// TwinCAT 3 PLC project FanucIntegrationV2
// ProgramVersion: 3.1.4026.26
// libraries:
//   Tc2_Standard, * (Beckhoff Automation GmbH)
//   Tc2_System, * (Beckhoff Automation GmbH)
//   FanucSimpleLib,2.1.0.0,Beckhoff Automation IL
// project tree:
//   DUTs/ E_FanucCstopiState.TcDUT, E_FanucEnableState.TcDUT, E_FanucFaultResetState.TcDUT, E_FanucHomingState.TcDUT, E_FanucStartProgramState.TcDUT, ST_FanucControl.TcDUT, ST_FanucStatus.TcDUT
//   GVLs/ GVL_Fanuc.TcGVL (not stored)
//   / PlcTask.TcTTO
//   POUs/ FB_FanucControl.TcPOU, FB_FanucCycleStop.TcPOU, FB_FanucEnable.TcPOU, FB_FanucFaultReset.TcPOU, FB_FanucHoming.TcPOU, FB_FanucSpeedOverride.TcPOU, FB_FanucStartProgram.TcPOU, FB_FanucStatus.TcPOU, MAIN.TcPOU
// real-time tasks:
//   TASK PlcTask: cycle T#10ms, priority 20, ADS port 350

CONFIGURATION FanucIntegrationV2
    RESOURCE PLC ON TwinCAT3
        TASK PlcTask(INTERVAL := T#10ms, PRIORITY := 20);
        PROGRAM MAIN WITH PlcTask : MAIN;
    END_RESOURCE
END_CONFIGURATION

// ---- DUTs/E_FanucCstopiState.TcDUT
// States used by FB_FanucCycleStop.

TYPE E_FanucCstopiState :
(
	Idle	:= 0, // Waits for a rising edge of bStart.
	Pulsing	:= 1, // Generates the CSTOPI pulse for tCycleStopPulse.
	Done	:= 2 // Sets bDone for one PLC scan to confirm pulse completion, then returns to Idle.
);
END_TYPE

// ---- DUTs/E_FanucEnableState.TcDUT
// States used by FB_FanucEnable.

TYPE E_FanucEnableState :
(
	Idle			:= 0, // ENBL is FALSE; waits for all enable permissives and bExtStart = FALSE.
	ClearFault		:= 1, // Waits for bFault = FALSE; this state does not generate FAULT_RESET.
	CheckTP			:= 3, // Waits for bTP_Enabled = FALSE before proceeding to WaitReady.
	WaitReady		:= 4, // Waits for bCmd_Enabled AND bSystem_Ready within tReadyTimeout.
	Ready			:= 5, // Sets bReady and accepts START edges while monitoring faults and interlocks.
	Paused			:= 6, // Waits for bExtHold = TRUE and bMotion_Held = FALSE before returning to Ready.
	EmergencyStop	:= 7, // Waits for bExtIMSTP = TRUE before returning through ClearFault.
	SafeSpeed		:= 8, // Waits for bExtSFSPD = TRUE before returning to Ready or Paused.
	Error			:= 99 // Sets bError and removes ENBL; bEnable = FALSE returns to Idle.
);
END_TYPE

// ---- DUTs/E_FanucFaultResetState.TcDUT
// States used by FB_FanucFaultReset.

TYPE E_FanucFaultResetState :
(
	Idle		:= 0, // Waits for a rising edge of bReset.
	SendPulse	:= 1, // Generates the FAULT_RESET pulse for tResetPulse.
	WaitClear	:= 2, // Waits for bFault = FALSE within tFaultTimeout after the pulse.
	Done		:= 3, // Sets bDone for one PLC scan, then returns to Idle.
	Error		:= 99 // Sets bError; bReset = FALSE returns to Idle.
);
END_TYPE

// ---- DUTs/E_FanucHomingState.TcDUT
// States used by FB_FanucHoming.

TYPE E_FanucHomingState :
(
	Idle			:= 0, // Waits for a rising edge of bStart while bReady = TRUE.
	RequestHome		:= 1, // Generates the HOME pulse for tHomePulse while bReady remains TRUE.
	WaitComplete	:= 2, // Waits for bAt_Home = TRUE within tHomingTimeout while bReady remains TRUE.
	Done			:= 3, // Sets bDone for one PLC scan, then returns to Idle.
	Error			:= 99 // Sets bError; bStart = FALSE returns to Idle.
);
END_TYPE

// ---- DUTs/E_FanucStartProgramState.TcDUT
// States used by FB_FanucStartProgram.

TYPE E_FanucStartProgramState :
(
	Idle	:= 0, // Waits for a rising edge of bStart while bReady = TRUE, then validates nProgram.
	Pulsing	:= 1, // Generates the selected RSR pulse for tProgramPulse and monitors its ACK.
	WaitAck	:= 2, // Waits for a fresh matching ACK within tAckTimeout after the pulse.
	Done	:= 3, // Sets bDone for one PLC scan to confirm acknowledgement, then returns to Idle.
	Error	:= 99 // Sets bError; bStart = FALSE returns to Idle.
);
END_TYPE

// ---- DUTs/ST_FanucControl.TcDUT
// FANUC command signals encoded by FB_FanucControl.
// UI numbers refer to robot inputs; aDO references refer to PLC output bytes.

TYPE ST_FanucControl :
STRUCT
	// Control byte 0: UI[1..8].
	IMSTP 		: BOOL; // aDO[0].0 | UI[1] *IMSTP: TRUE releases the request; FALSE requests an immediate stop.
	Hold		: BOOL; // aDO[0].1 | UI[2] *HOLD: TRUE releases the request; FALSE requests a hold.
	SFSPD		: BOOL; // aDO[0].2 | UI[3] *SFSPD: TRUE releases the request; FALSE asserts the SFSPD request.
	Cycle_stop	: BOOL; // aDO[0].3 | UI[4] CSTOPI: Cycle Stop command; effect depends on FANUC configuration.
	Fault_Reset	: BOOL; // aDO[0].4 | UI[5] FAULT_RESET: command pulse to reset clearable robot faults.
	Start		: BOOL; // aDO[0].5 | UI[6] START: start/resume command signal.
	Home		: BOOL; // aDO[0].6 | UI[7] HOME: command signal for the configured homing macro.
	Enable		: BOOL; // aDO[0].7 | UI[8] ENBL: TRUE enables motion subject to the remaining robot conditions.

	// Control byte 1: RSR selections or PNS bits, depending on robot mode.
	Start_Program1	: BOOL; // aDO[1].0 | UI[9]: RSR1 request or PNS bit 0.
	Start_Program2	: BOOL; // aDO[1].1 | UI[10]: RSR2 request or PNS bit 1.
	Start_Program3	: BOOL; // aDO[1].2 | UI[11]: RSR3 request or PNS bit 2.
	Start_Program4	: BOOL; // aDO[1].3 | UI[12]: RSR4 request or PNS bit 3.
	Start_Program5	: BOOL; // aDO[1].4 | UI[13]: RSR5 request or PNS bit 4.
	Start_Program6	: BOOL; // aDO[1].5 | UI[14]: RSR6 request or PNS bit 5.
	Start_Program7	: BOOL; // aDO[1].6 | UI[15]: RSR7 request or PNS bit 6.
	Start_Program8	: BOOL; // aDO[1].7 | UI[16]: RSR8 request or PNS bit 7.

	// Control byte 2: PNS command signals.
	PNS_Strobe	: BOOL; // aDO[2].0 | UI[17] PNSTROBE: strobe for PNS program selection.
	Prod_Start	: BOOL; // aDO[2].1 | UI[18] PROD_START: execution request for the selected PNS program.

	// Control byte 3: application-configured speed override.
	Override : BYTE; // aDO[3] | Speed-override command in percent; map to the configured FANUC Group Input.
END_STRUCT
END_TYPE

// ---- DUTs/ST_FanucStatus.TcDUT
// FANUC feedback signals decoded by FB_FanucStatus.
// UO numbers refer to robot outputs; aDI references refer to PLC input bytes.

TYPE ST_FanucStatus :
STRUCT
	// Status byte 0: UO[1..8].
	bCmd_Enabled	: BOOL; // aDI[0].0 | UO[1] CMDENBL: TRUE when the robot reports command enable.
	bSystem_Ready	: BOOL; // aDI[0].1 | UO[2] SYSRDY: TRUE when the robot reports system ready.
	bPrg_Running	: BOOL; // aDI[0].2 | UO[3] PROGRUN: TRUE when the robot reports program execution.
	bPrg_Paused		: BOOL; // aDI[0].3 | UO[4] PAUSED: TRUE when the robot reports a paused program.
	bMotion_Held	: BOOL; // aDI[0].4 | UO[5] HELD: TRUE when the robot reports motion held.
	bFault			: BOOL; // aDI[0].5 | UO[6] FAULT: TRUE when the robot reports a fault.
	bAt_Home		: BOOL; // aDI[0].6 | UO[7] ATPERCH: TRUE at the configured reference position used as Home.
	bTP_Enabled		: BOOL; // aDI[0].7 | UO[8] TPENBL: TRUE when the teach pendant is enabled.

	// Status byte 1: UO[9..10].
	bBatteryAlarm	: BOOL; // aDI[1].0 | UO[9] BATALM: TRUE when the robot reports a battery alarm.
	bBusy			: BOOL; // aDI[1].1 | UO[10] BUSY: robot busy indication; separate from individual FB busy outputs.

	// Status byte 2: RSR acknowledgements or PNS selection feedback.
	bProg_Start1ACK	: BOOL; // aDI[2].0 | UO[11]: RSR1 acknowledgement or SNO1 in PNS mode.
	bProg_Start2ACK	: BOOL; // aDI[2].1 | UO[12]: RSR2 acknowledgement or SNO2 in PNS mode.
	bProg_Start3ACK	: BOOL; // aDI[2].2 | UO[13]: RSR3 acknowledgement or SNO3 in PNS mode.
	bProg_Start4ACK	: BOOL; // aDI[2].3 | UO[14]: RSR4 acknowledgement or SNO4 in PNS mode.
	bProg_Start5ACK	: BOOL; // aDI[2].4 | UO[15]: RSR5 acknowledgement or SNO5 in PNS mode.
	bProg_Start6ACK	: BOOL; // aDI[2].5 | UO[16]: RSR6 acknowledgement or SNO6 in PNS mode.
	bProg_Start7ACK	: BOOL; // aDI[2].6 | UO[17]: RSR7 acknowledgement or SNO7 in PNS mode.
	bProg_Start8ACK	: BOOL; // aDI[2].7 | UO[18]: RSR8 acknowledgement or SNO8 in PNS mode.
END_STRUCT
END_TYPE

// ---- POUs/MAIN.TcPOU
PROGRAM MAIN
VAR
	// ---------- Core robot interface (library FBs) ----------
	fbStatus			: FB_FanucStatus;			// DI0 byte array → stStatus struct
	fbControl			: FB_FanucControl;			// stControl struct → DO0 byte array
	fbEnable			: FB_FanucEnable;			// Enable sequence state machine
	fbFaultReset		: FB_FanucFaultReset;		// Fault reset pulse – FAULT_RESET (UI[5])
	fbStartProgram		: FB_FanucStartProgram;		// Program start – RSR (UI[9..16])
	fbCycleStop			: FB_FanucCycleStop;		// Cycle Stop – CSTOPI (UI[4])
	fbHoming			: FB_FanucHoming;			// Homing sequence – HOME (UI[7])
	stStatus			: ST_FanucStatus;			// Live robot status (inputs)
	stControl			: ST_FanucControl;			// Combined control command (outputs)
	fbSpeedOverride		: FB_FanucSpeedOverride;	// Writes byOverwrite value to GI[25..33] via stControl

	// ---------- Enable command ----------
	bEnableRobot		: BOOL;	// Set TRUE to start enable sequence

	// ---------- External interlock signals ----------
	bExtIMSTP			: BOOL;		// Normally closed: FALSE = software E-stop
	bExtHold			: BOOL;		// Normally closed: FALSE = pause/hold robot
	bExtSFSPD			: BOOL;		// Normally closed: FALSE = safe-speed limit active
	bExtStart			: BOOL;		// Rising edge triggers a 20 ms START pulse when Ready

	// ---------- Homing ----------
	bStartHome			: BOOL;		// Rising edge: start homing sequence (gated by bReady)

	// ---------- Program start ----------
	bStartProgram		: BOOL;		// Rising edge: start nProgram (gated by bReady)
	nProgram			: INT := 1;	// Program to start: 1..8 (RSR)

	// ---------- Cycle stop ----------
	bCycleStop			: BOOL;		// Rising edge: send CSTOPI cycle-stop command

	// ---------- Fault reset ----------
	bFaultReset			: BOOL;		// Rising edge: send FAULT_RESET pulse (UI[5])

	// ---------- Speed override ----------
	byOverwrite			: BYTE;		// Value sent to GI[25..33] via fbSpeedOverride (0–100)
	
END_VAR

// 1. Read status – always first
fbStatus(aDI := GVL_Fanuc.DI0, stStatus => stStatus);

// 2. Enable sequence (outputs stControl; other FBs stamp into it below)
fbEnable(
    bEnable		:= bEnableRobot,
    stStatus	:= stStatus,
    bExtIMSTP	:= bExtIMSTP,   // Wire from: NOT bSoftEStop
    bExtHold	:= bExtHold,    // Wire from: NOT bPauseButton
    bExtSFSPD	:= bExtSFSPD,   // Wire from: bFenceOK / area scanner
    bExtStart 	:= bExtStart,   // Wire from: HMI start button
	tReadyTimeout := T#5S,
	bReady=> , 
	bError=> , 
	bTPWarning=> , 
	eState=> , 
    stControl => stControl);
	
// 3. Homing
fbHoming(
    bStart    := bStartHome,
    bReady    := fbEnable.bReady,
	tHomingTimeout := T#15S, 
    stStatus  := stStatus,
    stControl := stControl,
	bBusy=> , 
	bDone=> , 
	bError=> , 
	eState=> );
	
// 4. Program start 
fbStartProgram(
	bStart		:= bStartProgram, 
	nProgram	:= nProgram , 
	bReady		:= fbEnable.bReady, 
	tAckTimeout	:= T#2S , 
	stStatus	:= stStatus, 
	stControl	:= stControl, 
	bRequestActive=> , 
	bDone=> , 
	bError=> , 
	eState=> );
	
// 5. Cycle stop
fbCycleStop(
	bStart:= bCycleStop, 
	tCycleStopPulse:= T#20MS, 
	stControl:= stControl, 
	bBusy=> , 
	bDone=> , 
	eState=> );
	
// 6. Fault reset (call when fbEnable.eState = ClearFault and operator requests)
fbFaultReset(
    bReset    := bFaultReset,
    stStatus  := stStatus,
    stControl := stControl);

// 7. Control robot speed via Overwrite
fbSpeedOverride(
	nOverwrite:= byOverwrite ,
	stControl:= stControl ,
	bError=>,
	nActual=>);
	
// 8. Write outputs – always last
fbControl(aDO := GVL_Fanuc.DO0, stControl := stControl);

END_PROGRAM

// ---- POUs/FB_FanucStatus.TcPOU
// Maps the FANUC input bytes to robot-status signals.
// Call every PLC scan before status-dependent logic.

FUNCTION_BLOCK FB_FanucStatus

VAR_IN_OUT
	aDI : ARRAY[0..15] OF BYTE; // Hardware-linked input bytes; pass GVL_Fanuc.DI0. Reads bytes 0..2.
END_VAR

VAR_OUTPUT
	stStatus : ST_FanucStatus; // Robot-status signals decoded from aDI during this call.
END_VAR


// Status Byte 0  (aDI[0])  -  UO[1..8]
stStatus.bCmd_Enabled  := aDI[0].0;   // UO[1]  CMDENBL  – command enable
stStatus.bSystem_Ready := aDI[0].1;   // UO[2]  SYSRDY   – servo powered, no alarm
stStatus.bPrg_Running  := aDI[0].2;   // UO[3]  PROGRUN  – program in execution
stStatus.bPrg_Paused   := aDI[0].3;   // UO[4]  PAUSED   – program on hold
stStatus.bMotion_Held  := aDI[0].4;   // UO[5]  HELD     – HOLD button/signal active
stStatus.bFault        := aDI[0].5;   // UO[6]  FAULT    – alarm preventing execution
stStatus.bAt_Home      := aDI[0].6;   // UO[7]  ATPERCH  – robot at reference position 1
stStatus.bTP_Enabled   := aDI[0].7;   // UO[8]  TPENBL   – teach pendant enable switch ON

// Status Byte 1  (aDI[1])  -  UO[9..10]
stStatus.bBatteryAlarm := aDI[1].0;   // UO[9]  BATALM   – controller battery low
stStatus.bBusy         := aDI[1].1;   // UO[10] BUSY     – program executing or TP busy

// Status Byte 2  (aDI[2])  -  UO[11..18]  RSR ACK / SNO
stStatus.bProg_Start1ACK := aDI[2].0; // UO[11] ACK1/SNO1
stStatus.bProg_Start2ACK := aDI[2].1; // UO[12] ACK2/SNO2
stStatus.bProg_Start3ACK := aDI[2].2; // UO[13] ACK3/SNO3
stStatus.bProg_Start4ACK := aDI[2].3; // UO[14] ACK4/SNO4
stStatus.bProg_Start5ACK := aDI[2].4; // UO[15] ACK5/SNO5
stStatus.bProg_Start6ACK := aDI[2].5; // UO[16] ACK6/SNO6
stStatus.bProg_Start7ACK := aDI[2].6; // UO[17] ACK7/SNO7
stStatus.bProg_Start8ACK := aDI[2].7; // UO[18] ACK8/SNO8

END_FUNCTION_BLOCK

// ---- POUs/FB_FanucControl.TcPOU
// Maps the FANUC control signals to the output bytes.
// Call every PLC scan after all FANUC command FBs.

FUNCTION_BLOCK FB_FanucControl

VAR_IN_OUT
	aDO : ARRAY[0..15] OF BYTE; // Hardware-linked output bytes; pass GVL_Fanuc.DO0. Writes bytes 0..3.
END_VAR

VAR_INPUT
	stControl : ST_FanucControl; // Combined FANUC commands to encode into aDO.
END_VAR


// Control Byte 0  (aDO[0])  -  UI[1..8]
aDO[0].0 := stControl.IMSTP;        // UI[1]  *IMSTP       NC – hold TRUE; FALSE = software E-stop
aDO[0].1 := stControl.Hold;         // UI[2]  *HOLD        NC – hold TRUE; FALSE = decelerate & pause
aDO[0].2 := stControl.SFSPD;        // UI[3]  *SFSPD       NC – hold TRUE; FALSE = safe-speed limit
aDO[0].3 := stControl.Cycle_stop;   // UI[4]  CSTOPI       pulse to stop/abort current cycle
aDO[0].4 := stControl.Fault_Reset;  // UI[5]  FAULT_RESET  pulse to reset clearable alarms
aDO[0].5 := stControl.Start;        // UI[6]  START        falling-edge resumes paused program
aDO[0].6 := stControl.Home;         // UI[7]  HOME         macro use only
aDO[0].7 := stControl.Enable;       // UI[8]  ENBL         NC – hold TRUE; FALSE = disable all motion

// Control Byte 1  (aDO[1])  -  UI[9..16]  RSR / PNS
aDO[1].0 := stControl.Start_Program1; // UI[9]  RSR1 / PNS bit 0
aDO[1].1 := stControl.Start_Program2; // UI[10] RSR2 / PNS bit 1
aDO[1].2 := stControl.Start_Program3; // UI[11] RSR3 / PNS bit 2
aDO[1].3 := stControl.Start_Program4; // UI[12] RSR4 / PNS bit 3
aDO[1].4 := stControl.Start_Program5; // UI[13] RSR5 / PNS bit 4
aDO[1].5 := stControl.Start_Program6; // UI[14] RSR6 / PNS bit 5
aDO[1].6 := stControl.Start_Program7; // UI[15] RSR7 / PNS bit 6
aDO[1].7 := stControl.Start_Program8; // UI[16] RSR8 / PNS bit 7

// Control Byte 2  (aDO[2])  -  UI[17..18]
aDO[2].0 := stControl.PNS_Strobe;                   // UI[17] reserved
aDO[2].1 := stControl.Prod_Start;   // UI[18] PROD_START – triggers PNS program execution

// Control Byte 3  (aDO[3])  -  GI[25..33] user-defined output
aDO[3] := stControl.Override;

END_FUNCTION_BLOCK

// ---- POUs/FB_FanucEnable.TcPOU
// Controls the FANUC remote-enable sequence and START pulse.
// External IMSTP, HOLD, and SFSPD signals pass through in every state.
// Fault reset is handled separately by FB_FanucFaultReset.

FUNCTION_BLOCK FB_FanucEnable

VAR_INPUT
	bEnable		: BOOL; // TRUE requests enabling; FALSE returns the FB to Idle and clears its error.
	stStatus	: ST_FanucStatus; // Live robot-status signals from FB_FanucStatus.

	bExtIMSTP	: BOOL; // IMSTP permissive: TRUE releases the request; FALSE requests an immediate stop.
	bExtHold	: BOOL; // HOLD permissive: TRUE releases the request; FALSE requests a hold.
	bExtSFSPD	: BOOL; // SFSPD permissive: TRUE releases the request; FALSE asserts the SFSPD request.

	bExtStart	: BOOL; // Rising edge requests a START pulse while Ready; must be FALSE to begin enabling.
	tReadyTimeout	: TIME := T#5S; // Maximum time in WaitReady for bCmd_Enabled AND bSystem_Ready.
END_VAR

VAR_OUTPUT
	bReady		: BOOL; // TRUE while the enable state machine is in Ready.
	bError		: BOOL; // TRUE in Error after a ready timeout or invalid state; cleared by bEnable = FALSE.
	bTPWarning	: BOOL; // TRUE while in CheckTP and the teach pendant is enabled.
	eState		: E_FanucEnableState; // Current state exposed for diagnostics and HMI.
	stControl	: ST_FanucControl; // Control structure; this FB writes Enable, IMSTP, Hold, SFSPD, and Start.
END_VAR

VAR
	eCurrentState : E_FanucEnableState := E_FanucEnableState.Idle; // Internal state used by the sequence.
	bEnablePermissivesOk : BOOL; // TRUE when bEnable, bExtIMSTP, bExtHold, and bExtSFSPD are all TRUE.
	tonReadyTimeout : TON; // Measures the time spent waiting in WaitReady.
	rtExtStart : R_TRIG; // Detects the FALSE-to-TRUE transition of bExtStart.
	bStartPulseActive : BOOL; // Latches the START pulse until its timer expires or Ready is lost.
	tonStartPulse : TON; // Measures the active START pulse duration.
END_VAR

VAR CONSTANT
	tStartPulse : TIME := T#20MS; // Requested duration of the START output pulse on UI[6].
END_VAR

(*
    FB_FanucEnable

    Purpose
    -------
    Controls the FANUC remote-enable state machine and produces
    the required UI control signals.

    Enable sequence
    ---------------

        Idle
          |
          | bEnable
          | + all interlocks OK
          | + bExtStart released
          v
        ClearFault
          |
          | bFault = FALSE
          v
        CheckTP
          |
          | TP disabled
          v
        WaitReady
          |
          | CMDENBL + SYSRDY
          v
        Ready


    Enable permissives
    ------------------
    The enable sequence requires:

        bEnable
        bExtIMSTP
        bExtHold
        bExtSFSPD

    These are combined internally as:

        bEnablePermissivesOk

    bExtStart is NOT an enable permissive.

    Start is a momentary command and is handled independently.


    ClearFault
    ----------
    This FB does NOT generate FAULT_RESET.

    While bFault remains TRUE, the state remains ClearFault.

    Use FB_FanucFaultReset externally to reset the FANUC fault.
    Once stStatus.bFault becomes FALSE, this FB automatically
    proceeds to CheckTP.


    Start behavior
    --------------
    bExtStart must be FALSE before the enable sequence can begin.

    Once Ready, an actual FALSE -> TRUE edge of bExtStart generates
    a tStartPulse pulse on stControl.Start.

    A Start edge occurring before Ready is ignored.

    If bExtStart is already TRUE when the robot enters Ready,
    no Start pulse is generated. It must first return FALSE and
    then receive a new rising edge.


    NC signal behavior
    ------------------
    Option A: passive while disabled.

    Idle / Error:
        ENBL  = FALSE
        IMSTP = TRUE
        HOLD  = TRUE
        SFSPD = TRUE

    Active states:
        ENBL  = TRUE
        IMSTP = bExtIMSTP
        HOLD  = bExtHold
        SFSPD = bExtSFSPD


    Error reset
    -----------
    To leave Error:

        bEnable := FALSE

    The FB then returns to Idle. A subsequent TRUE starts a new
    enable sequence.
*)

// Enable permissives
// ============================================================================
//
// These signals determine whether the robot is allowed to proceed through
// the enable sequence.
//
// bExtStart is intentionally NOT included.
// Start is a command, not a permissive.
//
bEnablePermissivesOk := bEnable AND bExtIMSTP AND bExtHold AND bExtSFSPD;

// Start edge detection
// ============================================================================
//
// Detect the REAL external FALSE -> TRUE transition.
//
// Do not gate the R_TRIG input with the Ready state. Doing that can create
// an artificial rising edge when the state changes into Ready while
// bExtStart is already TRUE.

rtExtStart(CLK := bExtStart);

// Accept the edge only if we were already in Ready when the edge occurred.
//
// Because this is evaluated BEFORE the state machine, a Start edge occurring
// in WaitReady on the same scan that WaitReady -> Ready occurs is ignored.

IF rtExtStart.Q
   AND (eCurrentState = E_FanucEnableState.Ready) THEN
    bStartPulseActive := TRUE;
END_IF;


// Ready timeout
// ============================================================================
//
// Run the timeout only while waiting for the FANUC ready feedback.
//
tonReadyTimeout(
    IN := (eCurrentState = E_FanucEnableState.WaitReady),
    PT := tReadyTimeout
);

// State machine
// ============================================================================

CASE eCurrentState OF

    // IDLE ============================================================================
    E_FanucEnableState.Idle:

        (*Start the enable sequence only when:
        
         1. Enable has been requested
         2. All enable/interlock conditions are healthy
         3. Start is released
        
         Requiring Start to be released prevents an already-held Start
         command from being accepted when the robot becomes Ready.
        *)
		
        IF bEnablePermissivesOk
           AND NOT bExtStart THEN
            eCurrentState := E_FanucEnableState.ClearFault;
        END_IF;

    // CLEAR FAULT ============================================================================
    E_FanucEnableState.ClearFault:
	
        // Abort the enable sequence if any enable permissive is lost.
        IF NOT bEnablePermissivesOk THEN
            eCurrentState := E_FanucEnableState.Idle;
        // No FAULT_RESET pulse is generated here.
        // While bFault = TRUE, no transition occurs and the state therefore remains ClearFault.
        // FB_FanucFaultReset should clear the actual FANUC fault externally.

        ELSIF NOT stStatus.bFault THEN
            eCurrentState := E_FanucEnableState.CheckTP;
        END_IF;


    // CHECK TEACH PENDANT ============================================================================
    E_FanucEnableState.CheckTP:

        // Abort if the enable request or any startup interlock is lost.
        IF NOT bEnablePermissivesOk THEN
            eCurrentState := E_FanucEnableState.Idle;

        // TP must be disabled for remote operation.
        ELSIF NOT stStatus.bTP_Enabled THEN
            eCurrentState := E_FanucEnableState.WaitReady;
        END_IF;

    // WAIT FOR ROBOT READY ============================================================================
E_FanucEnableState.WaitReady:

    IF NOT bEnablePermissivesOk THEN
        eCurrentState:= E_FanucEnableState.Idle;

    // A FANUC fault has priority over becoming Ready.
    ELSIF stStatus.bFault THEN
        eCurrentState:= E_FanucEnableState.ClearFault;

    // TP must remain disabled for remote operation.
    ELSIF stStatus.bTP_Enabled THEN
        eCurrentState:= E_FanucEnableState.CheckTP;

    // Robot confirms remote command mode and system-ready.
    ELSIF stStatus.bCmd_Enabled AND stStatus.bSystem_Ready THEN
        eCurrentState:= E_FanucEnableState.Ready;

    // Robot failed to become ready within the configured timeout.
    ELSIF tonReadyTimeout.Q THEN
        eCurrentState:= E_FanucEnableState.Error;

    END_IF;

    // READY ============================================================================
    E_FanucEnableState.Ready:
        
		// Priority:
        // 1. Disable request
        // 2. FANUC fault
        // 3. Teach Pendant
        // 4. Emergency stop
        // 5. Safe speed
        // 6. Hold
        IF NOT bEnable THEN
            eCurrentState := E_FanucEnableState.Idle;

        ELSIF stStatus.bFault THEN
            eCurrentState := E_FanucEnableState.ClearFault;

        ELSIF stStatus.bTP_Enabled THEN
            eCurrentState := E_FanucEnableState.CheckTP;

        ELSIF NOT bExtIMSTP THEN
            eCurrentState := E_FanucEnableState.EmergencyStop;

        ELSIF NOT bExtSFSPD THEN
            eCurrentState := E_FanucEnableState.SafeSpeed;

        // Enter Paused immediately when the external HOLD is asserted.
        // bMotion_Held is also checked so that robot feedback can put us into Paused even if the hold originated elsewhere.
        ELSIF NOT bExtHold OR stStatus.bMotion_Held THEN
            eCurrentState := E_FanucEnableState.Paused;
        END_IF;

    // PAUSED / HOLD ============================================================================
    E_FanucEnableState.Paused:
        IF NOT bEnable THEN
            eCurrentState := E_FanucEnableState.Idle;

        ELSIF stStatus.bFault THEN
            eCurrentState := E_FanucEnableState.ClearFault;

        ELSIF stStatus.bTP_Enabled THEN
            eCurrentState := E_FanucEnableState.CheckTP;

        ELSIF NOT bExtIMSTP THEN
            eCurrentState := E_FanucEnableState.EmergencyStop;

        ELSIF NOT bExtSFSPD THEN
            eCurrentState := E_FanucEnableState.SafeSpeed;

        // Do not return to Ready just because bMotion_Held dropped.
        // The external HOLD request must ALSO be released.
        ELSIF bExtHold
              AND NOT stStatus.bMotion_Held THEN
            eCurrentState := E_FanucEnableState.Ready;
        END_IF;


    // EMERGENCY STOP ============================================================================
	E_FanucEnableState.EmergencyStop:
	
		// Remain here for as long as the external IMSTP request is active.
		IF NOT bEnable THEN
			eCurrentState:= E_FanucEnableState.Idle;

		// Once IMSTP is released, pass through ClearFault because
		// FANUC may require a fault reset before becoming Ready again.
		ELSIF bExtIMSTP THEN
			eCurrentState:= E_FanucEnableState.ClearFault;
			
		END_IF;

	// SAFE SPEED
	// ============================================================================
    E_FanucEnableState.SafeSpeed:
        IF NOT bEnable THEN
            eCurrentState := E_FanucEnableState.Idle;

        ELSIF stStatus.bFault THEN
            eCurrentState := E_FanucEnableState.ClearFault;

        ELSIF stStatus.bTP_Enabled THEN
            eCurrentState := E_FanucEnableState.CheckTP;

        ELSIF NOT bExtIMSTP THEN
            eCurrentState := E_FanucEnableState.EmergencyStop;

        // Safe-speed request released.
		ELSIF bExtSFSPD THEN
		
			IF NOT bExtHold OR stStatus.bMotion_Held THEN 
				eCurrentState:= E_FanucEnableState.Paused;
			ELSE
				eCurrentState:= E_FanucEnableState.Ready;
			END_IF;
		
		END_IF;

    // ERROR ============================================================================
    E_FanucEnableState.Error:

        // Error requires the enable request to be removed before another enable sequence can begin.
        IF NOT bEnable THEN
            eCurrentState := E_FanucEnableState.Idle;
        END_IF;

    // INVALID / UNKNOWN STATE ============================================================================
    ELSE
        eCurrentState := E_FanucEnableState.Error;
END_CASE;


// Cancel START pulse if Ready was lost
// ============================================================================
// This also handles a fault, TP enable, hold, E-stop, safe-speed request, disable request, etc. occurring during the 20 ms START pulse.
//
IF eCurrentState <> E_FanucEnableState.Ready THEN
    bStartPulseActive := FALSE;
END_IF;


// START pulse timer
// ============================================================================
// Once triggered, keep START asserted until tStartPulse has elapsed.
tonStartPulse(IN := bStartPulseActive, PT := tStartPulse);

// Clear the pulse latch once the pulse duration has elapsed.
IF tonStartPulse.Q THEN
    bStartPulseActive := FALSE;
END_IF;


// Derived FANUC control outputs
// ============================================================================

// ENBL is controlled by the enable state machine.
stControl.Enable := (eCurrentState <> E_FanucEnableState.Idle) AND (eCurrentState <> E_FanucEnableState.Error);

// External FANUC UOP requests are always passed through.
stControl.IMSTP := bExtIMSTP;
stControl.Hold  := bExtHold;
stControl.SFSPD := bExtSFSPD;

// START is only allowed while Ready.
stControl.Start := (eCurrentState = E_FanucEnableState.Ready) AND bStartPulseActive;

// Diagnostic outputs
// ============================================================================

eState := eCurrentState;

bReady := (eCurrentState = E_FanucEnableState.Ready);

bError := (eCurrentState = E_FanucEnableState.Error);

bTPWarning := (eCurrentState = E_FanucEnableState.CheckTP) AND stStatus.bTP_Enabled;

END_FUNCTION_BLOCK

// ---- POUs/FB_FanucFaultReset.TcPOU
// Pulses FAULT_RESET and confirms that the FANUC fault indication is FALSE.
// Call every PLC scan.

FUNCTION_BLOCK FB_FanucFaultReset

VAR_INPUT
	bReset			: BOOL; // Rising edge starts a reset request while Idle; FALSE clears the FB error.
	stStatus		: ST_FanucStatus; // Live robot-status signals from FB_FanucStatus.
	tFaultTimeout	: TIME := T#5S; // Maximum wait for bFault = FALSE after the reset pulse completes.
END_VAR

VAR_IN_OUT
	stControl : ST_FanucControl; // Shared FANUC control structure; this FB writes Fault_Reset only.
END_VAR

VAR_OUTPUT
	bBusy	: BOOL; // TRUE while in SendPulse or WaitClear.
	bDone	: BOOL; // TRUE for one PLC scan when the pulse is complete and bFault is FALSE.
	bError	: BOOL; // TRUE in Error after a fault-clear timeout or invalid state; cleared by bReset = FALSE.
	eState	: E_FanucFaultResetState; // Current state exposed for diagnostics and HMI.
END_VAR

VAR
	eCurrentState	: E_FanucFaultResetState := E_FanucFaultResetState.Idle; // Internal state used by the sequence.
	rtReset			: R_TRIG; // Detects the FALSE-to-TRUE transition of bReset.
	tonResetPulse	: TON; // Measures the FAULT_RESET pulse duration in SendPulse.
	tonFaultTimeout	: TON; // Measures the wait for bFault = FALSE in WaitClear.
END_VAR

VAR CONSTANT
	tResetPulse	: TIME := T#20MS; // Requested duration of the FAULT_RESET output pulse on UI[5].
END_VAR

// Reset edge detection
// ============================================================================
rtReset(CLK := bReset);

// State machine
// ============================================================================
CASE eCurrentState OF

    // IDLE
    // ========================================================================
    E_FanucFaultResetState.Idle:

        IF rtReset.Q THEN
            eCurrentState := E_FanucFaultResetState.SendPulse;
        END_IF;

    // SEND RESET PULSE
    // ========================================================================
    E_FanucFaultResetState.SendPulse:

        // Always complete the configured FAULT_RESET pulse.
        IF tonResetPulse.Q THEN
            // The fault may already have cleared during the pulse.
            IF NOT stStatus.bFault THEN
                eCurrentState := E_FanucFaultResetState.Done;
            ELSE
                eCurrentState := E_FanucFaultResetState.WaitClear;
            END_IF;

        END_IF;

    // WAIT FOR FAULT TO CLEAR
    // ========================================================================
    E_FanucFaultResetState.WaitClear:

        IF NOT stStatus.bFault THEN
            eCurrentState := E_FanucFaultResetState.Done;
        ELSIF tonFaultTimeout.Q THEN
            eCurrentState := E_FanucFaultResetState.Error;
        END_IF;

    // DONE
    // ========================================================================
    E_FanucFaultResetState.Done:

        // bDone is exposed for one PLC scan.
        eCurrentState := E_FanucFaultResetState.Idle;

    // ERROR
    // ========================================================================
    E_FanucFaultResetState.Error:

        // Require the reset request to be released before another attempt.
        IF NOT bReset THEN
            eCurrentState := E_FanucFaultResetState.Idle;
        END_IF;

    // INVALID / UNKNOWN STATE
    ELSE

        eCurrentState := E_FanucFaultResetState.Error;

END_CASE;

// Timers
// ============================================================================
// Each timer is called exactly once per PLC scan and is enabled only by
// its corresponding state.
tonResetPulse(
    IN := (eCurrentState = E_FanucFaultResetState.SendPulse),
    PT := tResetPulse
);

tonFaultTimeout(
    IN := (eCurrentState = E_FanucFaultResetState.WaitClear),
    PT := tFaultTimeout
);


// FANUC control output
// ============================================================================
// FAULT_RESET is asserted only while the pulse is active.
stControl.Fault_Reset := (eCurrentState = E_FanucFaultResetState.SendPulse) AND NOT tonResetPulse.Q;

// Diagnostic outputs
// ============================================================================
eState := eCurrentState;

bBusy := (eCurrentState = E_FanucFaultResetState.SendPulse) OR (eCurrentState = E_FanucFaultResetState.WaitClear);

bDone := (eCurrentState = E_FanucFaultResetState.Done);

bError := (eCurrentState = E_FanucFaultResetState.Error);

END_FUNCTION_BLOCK

// ---- POUs/FB_FanucStartProgram.TcPOU
// Pulses the selected RSR signal and waits for a fresh matching acknowledgement.
// Loss of bReady returns the FB to Idle without confirming the request.

FUNCTION_BLOCK FB_FanucStartProgram

VAR_INPUT
	bStart		: BOOL; // Rising edge starts a request while Idle and bReady; FALSE clears the FB error.
	nProgram	: INT; // Requested RSR selection, 1..8; latched when a valid request is accepted.
	bReady		: BOOL; // Enable permissive from FB_FanucEnable; must remain TRUE throughout the sequence.
	tAckTimeout	: TIME := T#2S; // Maximum additional wait for acknowledgement after the RSR pulse completes.
	stStatus	: ST_FanucStatus; // Live robot-status signals from FB_FanucStatus.
END_VAR

VAR_IN_OUT
	stControl	: ST_FanucControl; // Shared FANUC control structure; this FB writes Start_Program1..8 only.
END_VAR

VAR_OUTPUT
	bRequestActive	: BOOL; // TRUE while in Pulsing or WaitAck; does not indicate program execution.
	bDone			: BOOL; // TRUE for one PLC scan after the pulse completes and a fresh matching ACK is detected.
	bError			: BOOL; // TRUE in Error after invalid selection, ACK timeout, or invalid state; cleared by bStart = FALSE.
	eState			: E_FanucStartProgramState; // Current state exposed for diagnostics and HMI.
END_VAR

VAR
	eCurrentState	: E_FanucStartProgramState := E_FanucStartProgramState.Idle; // Internal state used by the sequence.
	rtStart			: R_TRIG; // Detects the FALSE-to-TRUE transition of bStart.
	nActiveProgram	: INT; // Latched RSR selection used for the active output and matching ACK.
	bActiveAck		: BOOL; // Current acknowledgement signal corresponding to nActiveProgram.
	bAckArmed		: BOOL; // TRUE once the selected ACK has been observed FALSE during the active sequence.
	bAckSeen		: BOOL; // Latched TRUE when the selected ACK is TRUE after acknowledgement detection is armed.
	bRsrPulseActive	: BOOL; // TRUE while the selected RSR output pulse is active.
	tonProgramPulse	: TON; // Measures the selected RSR pulse duration in Pulsing.
	tonAckTimeout	: TON; // Measures the additional acknowledgement wait in WaitAck.
END_VAR

VAR CONSTANT
	tProgramPulse : TIME := T#200MS; // Requested duration of the selected RSR output pulse on UI[9..16].
END_VAR

// Start edge detection
// ============================================================================
rtStart(CLK := bStart);

// Latch a valid program selection before reading its ACK
// ============================================================================
// This allows the Idle state to inspect the newly selected ACK before
// asserting the RSR output during this PLC scan.

IF (eCurrentState = E_FanucStartProgramState.Idle) AND rtStart.Q AND bReady AND (nProgram >= 1) AND (nProgram <= 8) THEN
	nActiveProgram := nProgram;
END_IF;


// Selected acknowledgement
// ============================================================================
CASE nActiveProgram OF

	1: bActiveAck := stStatus.bProg_Start1ACK;
	2: bActiveAck := stStatus.bProg_Start2ACK;
	3: bActiveAck := stStatus.bProg_Start3ACK;
	4: bActiveAck := stStatus.bProg_Start4ACK;
	5: bActiveAck := stStatus.bProg_Start5ACK;
	6: bActiveAck := stStatus.bProg_Start6ACK;
	7: bActiveAck := stStatus.bProg_Start7ACK;
	8: bActiveAck := stStatus.bProg_Start8ACK;

ELSE
	bActiveAck := FALSE;

END_CASE;


// Acknowledgement detection
// ============================================================================
// Remember a fresh ACK received during either the pulse or the ACK wait.
// An ACK already HIGH when the request is accepted must first become LOW.

IF (eCurrentState = E_FanucStartProgramState.Pulsing) OR (eCurrentState = E_FanucStartProgramState.WaitAck) THEN

	IF NOT bActiveAck THEN
		bAckArmed := TRUE;
	END_IF;

	IF bAckArmed AND bActiveAck THEN
		bAckSeen := TRUE;
	END_IF;

END_IF;

// State machine
// ============================================================================
CASE eCurrentState OF

	// IDLE
	// ========================================================================
	E_FanucStartProgramState.Idle:
	
		IF rtStart.Q AND bReady THEN
			IF (nProgram < 1) OR (nProgram > 8) THEN
				eCurrentState := E_FanucStartProgramState.Error;
			ELSE
				// nActiveProgram and its matching ACK were selected above.
				// Arm immediately if ACK is LOW before RSR is asserted.
				bAckArmed := NOT bActiveAck;
				bAckSeen := FALSE;

				eCurrentState := E_FanucStartProgramState.Pulsing;
			END_IF;
		END_IF;


	// PULSING
	// ========================================================================
	E_FanucStartProgramState.Pulsing:
	
		IF NOT bReady THEN
			eCurrentState := E_FanucStartProgramState.Idle;
		ELSIF tonProgramPulse.Q THEN
			// Complete the pulse even if ACK arrived before it ended.
			IF bAckSeen THEN
				eCurrentState := E_FanucStartProgramState.Done;
			ELSE
				eCurrentState := E_FanucStartProgramState.WaitAck;
			END_IF;
		END_IF;

	// WAIT FOR ACKNOWLEDGEMENT
	// ========================================================================
	E_FanucStartProgramState.WaitAck:

		IF NOT bReady THEN
			eCurrentState := E_FanucStartProgramState.Idle;
		ELSIF bAckSeen THEN
			eCurrentState := E_FanucStartProgramState.Done;
		ELSIF tonAckTimeout.Q THEN
			eCurrentState := E_FanucStartProgramState.Error;
		END_IF;

	// DONE
	// ========================================================================
	E_FanucStartProgramState.Done:

		// The Done state is exposed for one PLC scan.
		eCurrentState := E_FanucStartProgramState.Idle;

	// ERROR
	// ========================================================================
	E_FanucStartProgramState.Error:

		// Release Start before another request can be accepted.
		IF NOT bStart THEN
			eCurrentState := E_FanucStartProgramState.Idle;
		END_IF;

	// INVALID / UNKNOWN STATE
	// ========================================================================
	ELSE
		eCurrentState := E_FanucStartProgramState.Error;
END_CASE;


// Timers
// ============================================================================
// Each timer is called once per scan and enabled by its corresponding state.

tonProgramPulse(
	IN := (eCurrentState = E_FanucStartProgramState.Pulsing),
	PT := tProgramPulse
);

tonAckTimeout(
	IN := (eCurrentState = E_FanucStartProgramState.WaitAck),
	PT := tAckTimeout
);


// Clear handshake flags while Idle
// ============================================================================
IF eCurrentState = E_FanucStartProgramState.Idle THEN

	bAckArmed := FALSE;
	bAckSeen := FALSE;

END_IF;


// FANUC RSR control outputs
// ============================================================================
// Assign every RSR output once per scan.
// Only the selected output can be TRUE while the pulse is active.

bRsrPulseActive := (eCurrentState = E_FanucStartProgramState.Pulsing) AND NOT tonProgramPulse.Q;

stControl.Start_Program1 := bRsrPulseActive AND (nActiveProgram = 1);
stControl.Start_Program2 := bRsrPulseActive AND (nActiveProgram = 2);
stControl.Start_Program3 := bRsrPulseActive AND (nActiveProgram = 3);
stControl.Start_Program4 := bRsrPulseActive AND (nActiveProgram = 4);
stControl.Start_Program5 := bRsrPulseActive AND (nActiveProgram = 5);
stControl.Start_Program6 := bRsrPulseActive AND (nActiveProgram = 6);
stControl.Start_Program7 := bRsrPulseActive AND (nActiveProgram = 7);
stControl.Start_Program8 := bRsrPulseActive AND (nActiveProgram = 8);


// Diagnostic outputs
// ============================================================================
eState := eCurrentState;

bRequestActive := (eCurrentState = E_FanucStartProgramState.Pulsing) OR (eCurrentState = E_FanucStartProgramState.WaitAck);

bDone := (eCurrentState = E_FanucStartProgramState.Done);

bError := (eCurrentState = E_FanucStartProgramState.Error);

END_FUNCTION_BLOCK

// ---- POUs/FB_FanucCycleStop.TcPOU
// Pulses CSTOPI; the FANUC "CSTOPI for ABORT" setting determines its effect.
// Completion confirms the output pulse only; no robot acknowledgement is checked.

FUNCTION_BLOCK FB_FanucCycleStop

VAR_INPUT
	bStart			: BOOL; // Rising edge starts a Cycle Stop request while Idle.
	tCycleStopPulse	: TIME := T#20MS; // Requested duration of the CSTOPI output pulse on UI[4].
END_VAR

VAR_IN_OUT
	stControl	: ST_FanucControl; // Shared FANUC control structure; this FB writes Cycle_stop only.
END_VAR

VAR_OUTPUT
	bBusy	: BOOL; // TRUE while the sequence is in Pulsing.
	bDone	: BOOL; // TRUE for one PLC scan after the pulse completes; does not confirm stopped motion.
	eState	: E_FanucCstopiState; // Current state exposed for diagnostics and HMI.
END_VAR

VAR
	eCurrentState		: E_FanucCstopiState := E_FanucCstopiState.Idle; // Internal state used by the sequence.
	rtStart				: R_TRIG; // Detects the FALSE-to-TRUE transition of bStart.
	tonCycleStopPulse	: TON; // Measures the CSTOPI pulse duration in Pulsing.
END_VAR

// Start edge detection
// ============================================================================
rtStart(CLK := bStart);

// State machine
// ============================================================================
CASE eCurrentState OF

    // IDLE
    // ========================================================================
    E_FanucCstopiState.Idle:

        IF rtStart.Q THEN
            eCurrentState := E_FanucCstopiState.Pulsing;
        END_IF;

    // PULSING
    // ========================================================================
    E_FanucCstopiState.Pulsing:

        IF tonCycleStopPulse.Q THEN
            eCurrentState := E_FanucCstopiState.Done;
        END_IF;

    // DONE
    // ========================================================================
    E_FanucCstopiState.Done:

        // bDone is exposed for one PLC scan.
        eCurrentState := E_FanucCstopiState.Idle;

    // INVALID / UNKNOWN STATE
    // ========================================================================
    ELSE

        // Cycle Stop has no error-recovery sequence.
        // Return safely to Idle and remove CSTOPI.
        eCurrentState := E_FanucCstopiState.Idle;

END_CASE;

// Cycle Stop pulse timer
// ============================================================================
// The timer is called exactly once per PLC scan.

tonCycleStopPulse(
    IN := (eCurrentState = E_FanucCstopiState.Pulsing),
    PT := tCycleStopPulse
);

// FANUC control output
// ============================================================================
// CSTOPI is asserted only while the pulse is active.

stControl.Cycle_stop :=
    (eCurrentState = E_FanucCstopiState.Pulsing) AND NOT tonCycleStopPulse.Q;

// Diagnostic outputs
// ============================================================================
eState := eCurrentState;

bBusy := (eCurrentState = E_FanucCstopiState.Pulsing);

bDone := (eCurrentState = E_FanucCstopiState.Done);

END_FUNCTION_BLOCK

// ---- POUs/FB_FanucHoming.TcPOU
// Pulses HOME and waits for the configured home-position feedback.
// Loss of bReady returns the FB to Idle without confirming completion.

FUNCTION_BLOCK FB_FanucHoming

VAR_INPUT
	bStart			: BOOL; // Rising edge starts homing while Idle and bReady; FALSE clears the FB error.
	bReady			: BOOL; // Enable permissive from FB_FanucEnable; must remain TRUE throughout the sequence.
	tHomingTimeout	: TIME := T#30S; // Maximum wait for bAt_Home = TRUE after the HOME pulse completes.
	stStatus		: ST_FanucStatus; // Live robot-status signals from FB_FanucStatus.
END_VAR

VAR_IN_OUT
	stControl	: ST_FanucControl; // Shared FANUC control structure; this FB writes Home only.
END_VAR

VAR_OUTPUT
	bBusy	: BOOL; // TRUE while in RequestHome or WaitComplete.
	bDone	: BOOL; // TRUE for one PLC scan when bAt_Home is TRUE in WaitComplete.
	bError	: BOOL; // TRUE in Error after a homing timeout or invalid state; cleared by bStart = FALSE.
	eState	: E_FanucHomingState; // Current state exposed for diagnostics and HMI.
END_VAR

VAR
	eCurrentState		: E_FanucHomingState := E_FanucHomingState.Idle; // Internal state used by the sequence.
	rtStart				: R_TRIG; // Detects the FALSE-to-TRUE transition of bStart.
	tonHomePulse		: TON; // Measures the HOME pulse duration in RequestHome.
	tonHomingTimeout	: TON; // Measures the wait for bAt_Home = TRUE in WaitComplete.
END_VAR

VAR CONSTANT
	tHomePulse	: TIME := T#200MS; // Requested duration of the HOME output pulse on UI[7].
END_VAR

(*
    FB_FanucHoming

    Purpose
    -------
    Controls the FANUC homing sequence and generates the HOME (UI[7])
    command used to trigger the configured homing macro or program.


    Homing sequence
    ---------------

        Idle
          |
          | bStart rising edge
          | + bReady
          v
        RequestHome
          |
          | HOME asserted for tHomePulse
          v
        WaitComplete
          |
          | bAt_Home = TRUE
          v
        Done
          |
          | one PLC scan
          v
        Idle


    Start behavior
    --------------
    bStart is treated as a momentary command.

    The R_TRIG detects the actual external FALSE -> TRUE transition:

        rtStart(CLK := bStart);

    The edge is accepted only when:

        bReady = TRUE
        AND
        eCurrentState = Idle

    A Start edge occurring while the robot is not Ready is ignored.

    If bStart goes TRUE before bReady becomes TRUE and remains TRUE,
    becoming Ready must NOT automatically start homing.

    bStart must first return FALSE and then receive a new rising edge.


    HOME pulse
    ----------
    RequestHome represents the HOME command pulse state.

    While RequestHome is active:

        stControl.Home = TRUE

    The HOME signal remains asserted for:

        tHomePulse

    After the pulse completes, the FB transitions to WaitComplete.


    Homing completion
    -----------------
    While in WaitComplete, the FB waits for:

        stStatus.bAt_Home = TRUE

    Once confirmed, the FB transitions to Done.

    bDone is TRUE for one PLC scan before the state returns to Idle.


    Ready interlock
    ---------------
    Homing may only start while:

        bReady = TRUE

    If bReady becomes FALSE during RequestHome or WaitComplete,
    the FB stops considering the homing sequence valid and returns
    to Idle.

    Returning this FB to Idle does not necessarily cancel a FANUC
    program or macro that has already started. Actual robot stopping
    behavior is controlled by the FANUC controller and its other UOP
    control inputs.


    Timeout
    -------
    While in WaitComplete, tonHomingTimeout runs for:

        tHomingTimeout

    If bAt_Home is not confirmed before the timeout expires,
    the FB transitions to Error.


    Error reset
    -----------
    To leave Error:

        bStart := FALSE

    The FB then returns to Idle.

    A new FALSE -> TRUE edge of bStart is required before another
    homing sequence can begin.


    FANUC prerequisites
    -------------------
    - HOME (UI[7]) must be configured to trigger the required
      homing macro or program.

    - stStatus.bAt_Home must represent the FANUC home-position
      feedback used by the application.


    Usage
    -----
    - Call this FB every PLC cycle.

    - Wire bReady from:

          FB_FanucEnable.bReady

    - Pass the same stControl instance used by the other FANUC
      command FBs and by FB_FanucControl.

    - Generate a rising edge on bStart to request homing.

    - Monitor:

          bBusy
          bDone
          bError
          eState
*)

// Start edge detection
// ============================================================================
//
// Detect the real external FALSE -> TRUE transition.
// Do not gate R_TRIG with bReady.
//
rtStart(CLK := bStart);

// State machine
// ============================================================================

CASE eCurrentState OF

    // IDLE ====================================================================
    E_FanucHomingState.Idle:

        // Accept Home only if the rising edge occurs while robot is Ready.
        IF rtStart.Q AND bReady THEN
            eCurrentState := E_FanucHomingState.RequestHome;
        END_IF;


    // REQUEST HOME ============================================================
    E_FanucHomingState.RequestHome:

        // Abort this FB sequence if robot Ready is lost.
        IF NOT bReady THEN
            eCurrentState := E_FanucHomingState.Idle;
        // HOME pulse completed.
        ELSIF tonHomePulse.Q THEN
            eCurrentState := E_FanucHomingState.WaitComplete;
        END_IF;

    // WAIT FOR HOME ===========================================================
    E_FanucHomingState.WaitComplete:

        IF NOT bReady THEN
            eCurrentState := E_FanucHomingState.Idle;
        // FANUC confirms Home position.
        ELSIF stStatus.bAt_Home THEN
            eCurrentState := E_FanucHomingState.Done;
        // Homing did not complete in time.
        ELSIF tonHomingTimeout.Q THEN
            eCurrentState := E_FanucHomingState.Error;
        END_IF;


    // DONE ====================================================================
    E_FanucHomingState.Done:

        // Done is exposed for one PLC scan.
        eCurrentState := E_FanucHomingState.Idle;

    // ERROR ===================================================================
    E_FanucHomingState.Error:

        // Require Start to be released before allowing another attempt.
        IF NOT bStart THEN
            eCurrentState := E_FanucHomingState.Idle;
        END_IF;

    // INVALID / UNKNOWN STATE =================================================
    ELSE
        eCurrentState := E_FanucHomingState.Error;
END_CASE;


// Timers
// ============================================================================
//
// Timers are enabled only by their corresponding state.

tonHomePulse(
    IN := (eCurrentState = E_FanucHomingState.RequestHome),
    PT := tHomePulse
);

tonHomingTimeout(
    IN := (eCurrentState = E_FanucHomingState.WaitComplete),
    PT := tHomingTimeout
);


// Derived FANUC control output
// ============================================================================
//
// HOME is asserted only during RequestHome and drops as soon as the
// configured pulse time has elapsed.

stControl.Home := (eCurrentState = E_FanucHomingState.RequestHome) AND NOT tonHomePulse.Q;

// Diagnostic outputs
// ============================================================================

eState := eCurrentState;

bBusy := (eCurrentState = E_FanucHomingState.RequestHome) OR (eCurrentState = E_FanucHomingState.WaitComplete);

bDone := (eCurrentState = E_FanucHomingState.Done);

bError := (eCurrentState = E_FanucHomingState.Error);

END_FUNCTION_BLOCK

// ---- POUs/FB_FanucSpeedOverride.TcPOU
// Continuously writes the validated speed-override command.
// Values above 100 produce a 0% command and set bError.

FUNCTION_BLOCK FB_FanucSpeedOverride

VAR_INPUT
	nOverwrite	: BYTE; // Requested speed override in percent; valid range: 0..100.
END_VAR

VAR_IN_OUT
	stControl	: ST_FanucControl; // Shared FANUC control structure; this FB writes Overwrite only.
END_VAR

VAR_OUTPUT
	bError	: BOOL; // TRUE while nOverwrite exceeds cMaxOverwrite; clears when the input becomes valid.
	nActual	: BYTE; // Override command written to stControl.Overwrite; not robot feedback. Invalid input produces 0.
END_VAR

VAR CONSTANT
	cMaxOverwrite	: BYTE := 100; // Maximum accepted speed-override command in percent.
END_VAR

// Input validation
// ============================================================================
bError := nOverwrite > cMaxOverwrite;

// Determine actual output value
// ============================================================================
// An invalid value results in 0% override.
//
// This keeps the result deterministic and prevents an invalid command
// from leaving the previous overwrite value active.

IF bError THEN
    nActual := 0;
ELSE
    nActual := nOverwrite;
END_IF;


// FANUC control output
// ============================================================================
// Continuously write the validated overwrite value to the shared
// FANUC control structure.

stControl.Override := nActual;

END_FUNCTION_BLOCK
